(* PLC project Unnamed, Unknown Unnamed 1 *)
(* stored: creationDateTime 2024-03-25T14:39:34, modificationDateTime 2024-03-27T15:07:07 *)

PROGRAM aqua_sys
  VAR
    low_DO AT %QX0.0 : BOOL;
    high_DO AT %QX0.1 : BOOL;
    airpump AT %QX0.2 : BOOL;
    pH AT %QX0.3 : BOOL;
    pHalert AT %QX0.4 : BOOL;
    low_temp AT %QX0.5 : BOOL;
    high_temp AT %QX0.6 : BOOL;
    heating AT %QX0.7 : BOOL;
    waterpump AT %QX1.0 : BOOL;
    wp_on AT %QX1.1 : BOOL;
    wp_off AT %QX1.2 : BOOL;
    wplatched AT %QX1.3 : BOOL;
  END_VAR

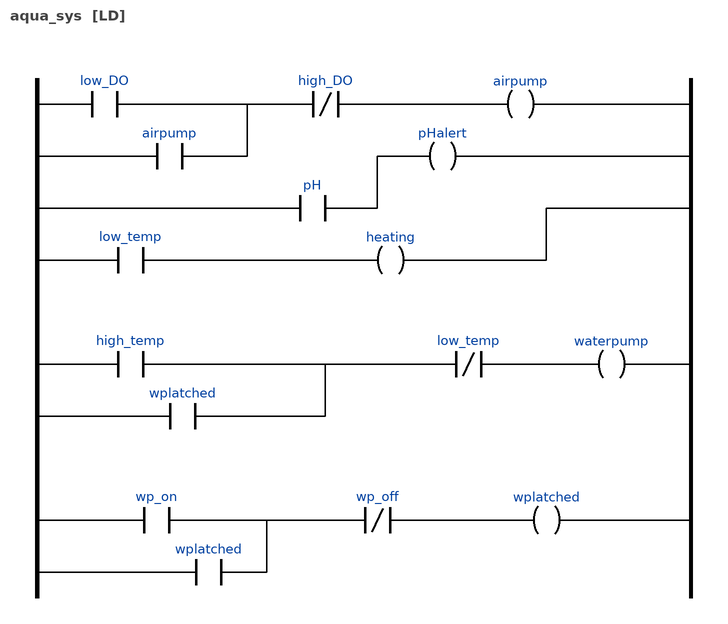
(* LD diagram, written out as Structured Text *)
airpump := (low_DO OR airpump) AND NOT high_DO;
pHalert := pH;
heating := low_temp;
waterpump := (high_temp OR wplatched) AND NOT low_temp;
wplatched := (wp_on OR wplatched) AND NOT wp_off;
END_PROGRAM

CONFIGURATION Config0
  RESOURCE Res0 ON PLC
    TASK task0(INTERVAL := T#20ms, PRIORITY := 0);
    PROGRAM instance0 WITH task0 : aqua_sys;
  END_RESOURCE
END_CONFIGURATION
